// TIA Portal V17 export
// export: Created 2024-09-02T12:50:40.2797214Z, ExportSetting WithDefaults, DisplayName Totally Integrated Automation Portal, DisplayVersion V17, DisplayName TIA Portal Openness, DisplayVersion V17, DisplayName TIA Portal Version Control Interface, DisplayVersion V17, DisplayName STEP 7 Professional, DisplayVersion V17, DisplayName STEP 7 Safety, DisplayVersion V17, DisplayName WinCC Professional, DisplayVersion V17
TYPE "Scania_typ_General"
// stored: IsFailsafeCompliant false
   STRUCT
      "Pallet Number" : Int;
      "HA ID" : String[16];
      ID : String[16];   // only for LS, IS, GS
      Variant : String[32];
      "POP ID" : String[16];
      VariantCode : Int;
      "Pallet Status" : Struct
         "Pallet loaded" : Bool;
         "Global NOK" : Bool;
         Bypass : Bool;
         Repaired : Bool;
         Scraped : Bool;
         "Sequence healing" : Bool;
         "Plan B" : Bool;
         "Master pallet" : Bool;
         "Res byte" : Byte;
      END_STRUCT;
      "NOK Code number" : Int;
      Measurement : Struct
         "HA1.7" : Struct
            "Bearing65/69.86" : Struct
               MeasuredValue : Real;
               MinValue : Real;
               MaxValue : Real;
            END_STRUCT;
            Bearing65 : Struct
               MeasuredValue : Real;
               MinValue : Real;
               MaxValue : Real;
            END_STRUCT;
         END_STRUCT;
         "HA2.4" : Struct
            FrontBearing : Struct
               MeasuredValue : Real;
               MinValue : Real;
               MaxValue : Real;
            END_STRUCT;
            HightOfFrontBearing : Struct
               MeasuredValue : Real;
               MinValue : Real;
               MaxValue : Real;
            END_STRUCT;
            RearBearing : Struct
               MeasuredValue : Real;
               MinValue : Real;
               MaxValue : Real;
            END_STRUCT;
            HightOfRearBearing : Struct
               MeasuredValue : Real;
               MinValue : Real;
               MaxValue : Real;
            END_STRUCT;
            HightZSB : Struct
               MeasuredValue : Real;
               MinValue : Real;
               MaxValue : Real;
            END_STRUCT;
         END_STRUCT;
         "HA2.6" : Struct
            Shim : Struct
               MeasuredValue : Real;
               MinValue : Real;
               MaxValue : Real;
            END_STRUCT;
         END_STRUCT;
      END_STRUCT;
      Reserve : Array[88..99] of Byte;
   END_STRUCT;
END_TYPE
